(* Logix 5000 project; controller cal1632 1756-L62 rev 16.20; software revision 16.05; part 32 of 61 *)
(* tags used below, declared in another part *)
   FAULT : BOOL;
   HMI : BOOL;
   p01_recipe_active : recipe;
   p01r09 : routine;
   p01r09_pb_global_reset : BOOL;
   p01r13_line_running : BOOL;
   p02_dint_from_hmi : hmi_dint;
   p20_di_acc_empty : BOOL;
   p20_do_close_nip : BOOL;
   p20_do_engage_lfr_clutch : BOOL;
   p21_di_close_exit_clamp : BOOL;
   p21_di_close_inlet_clamp : BOOL;
   p21_di_open_splice_platen : BOOL;
   p21_di_platen_not_closed : BOOL;
   p21_di_splice_2_hand_close : BOOL;
   p21_dint_to_hmi : DINT[16];
   p21_do_close_exit_clamp_sv : BOOL;
   p21_do_close_inlet_clamp_sv : BOOL;
   p21_do_close_platen_sv : BOOL;
   p21r07 : routine;
   p21r07_timer_fault : TIMER[4];
   p21r07_timer_warning : TIMER[4];
   p21r08 : routine;
   p21r08_timer_fault : TIMER[4];
   p21r08_timer_warning : TIMER[4];
   p21r09 : routine;
   p21r09_timer_fault : TIMER[4];
   p21r09_timer_warning : TIMER[4];
   p21r10 : routine;
   p21r10_permissive_run : BOOL;
   p21r10_remaining_cure_time : DINT;
   p21r10_remaining_cure_time_sec : REAL;
   p21r10_splice_press_1 : SYS_ENC;
   p21r10_state : DINT;
   p21r10_status : DINT;
   p21r10_timer_exit_open_delay : TIMER;
   p21r10_timer_fault : TIMER[4];
   p21r10_timer_inlet_open_delay : TIMER;
   p21r10_timer_platen_open_delay : TIMER;
   p21r10_timer_press_cure : TIMER;
   p21r10_timer_warning : TIMER[4];
   p21r16 : routine;
(* P21_Splice_Press, continued *)

ROUTINE R07_Alarms   (* ladder *)
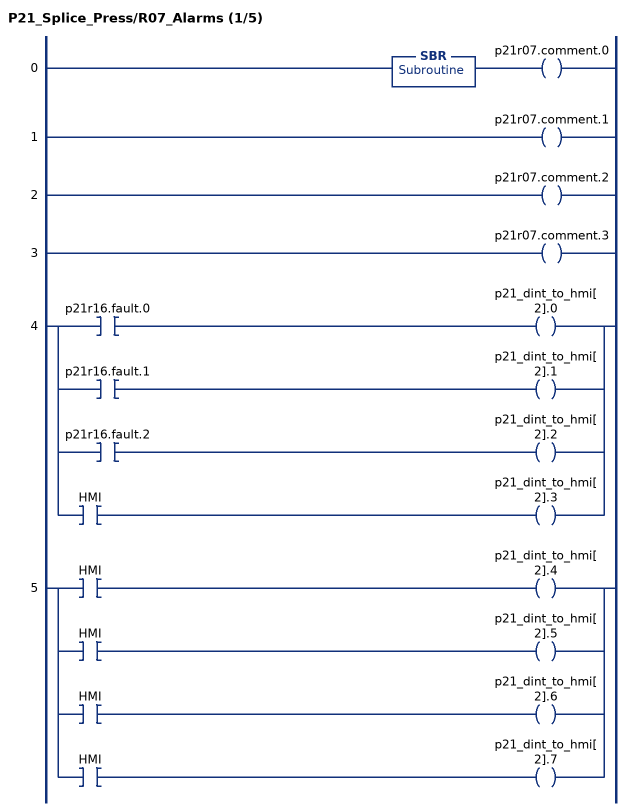
   0: SBR()OTE(p21r07.comment.0);
   1: OTE(p21r07.comment.1);
   2: OTE(p21r07.comment.2);
   3: OTE(p21r07.comment.3);
   4: [XIC(p21r16.fault.0) OTE(p21_dint_to_hmi[2].0) ,XIC(p21r16.fault.1) OTE(p21_dint_to_hmi[2].1) ,XIC(p21r16.fault.2) OTE(p21_dint_to_hmi[2].2) ,XIC(HMI) OTE(p21_dint_to_hmi[2].3) ];
   5: [XIC(HMI) OTE(p21_dint_to_hmi[2].4) ,XIC(HMI) OTE(p21_dint_to_hmi[2].5) ,XIC(HMI) OTE(p21_dint_to_hmi[2].6) ,XIC(HMI) OTE(p21_dint_to_hmi[2].7) ];
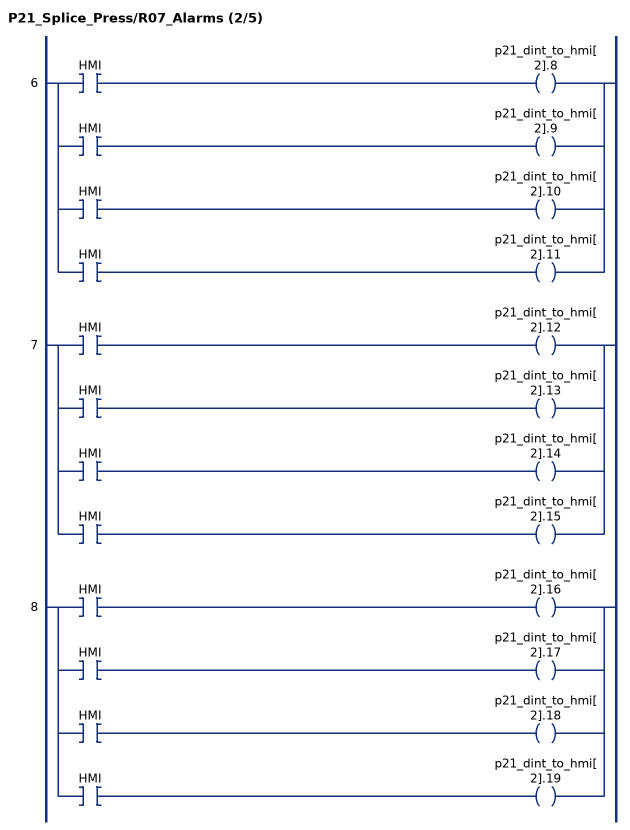
   6: [XIC(HMI) OTE(p21_dint_to_hmi[2].8) ,XIC(HMI) OTE(p21_dint_to_hmi[2].9) ,XIC(HMI) OTE(p21_dint_to_hmi[2].10) ,XIC(HMI) OTE(p21_dint_to_hmi[2].11) ];
   7: [XIC(HMI) OTE(p21_dint_to_hmi[2].12) ,XIC(HMI) OTE(p21_dint_to_hmi[2].13) ,XIC(HMI) OTE(p21_dint_to_hmi[2].14) ,XIC(HMI) OTE(p21_dint_to_hmi[2].15) ];
   8: [XIC(HMI) OTE(p21_dint_to_hmi[2].16) ,XIC(HMI) OTE(p21_dint_to_hmi[2].17) ,XIC(HMI) OTE(p21_dint_to_hmi[2].18) ,XIC(HMI) OTE(p21_dint_to_hmi[2].19) ];
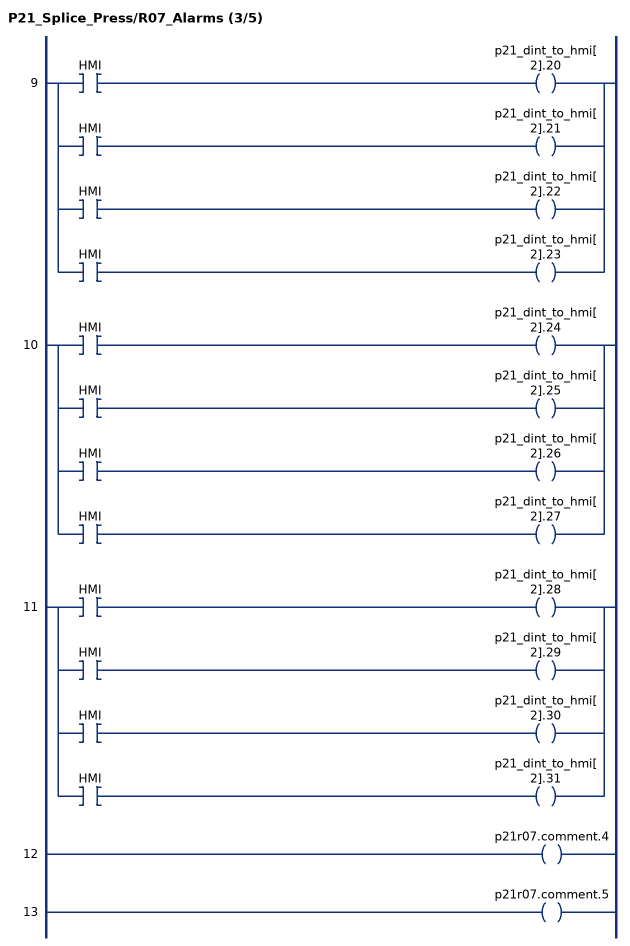
   9: [XIC(HMI) OTE(p21_dint_to_hmi[2].20) ,XIC(HMI) OTE(p21_dint_to_hmi[2].21) ,XIC(HMI) OTE(p21_dint_to_hmi[2].22) ,XIC(HMI) OTE(p21_dint_to_hmi[2].23) ];
   10: [XIC(HMI) OTE(p21_dint_to_hmi[2].24) ,XIC(HMI) OTE(p21_dint_to_hmi[2].25) ,XIC(HMI) OTE(p21_dint_to_hmi[2].26) ,XIC(HMI) OTE(p21_dint_to_hmi[2].27) ];
   11: [XIC(HMI) OTE(p21_dint_to_hmi[2].28) ,XIC(HMI) OTE(p21_dint_to_hmi[2].29) ,XIC(HMI) OTE(p21_dint_to_hmi[2].30) ,XIC(HMI) OTE(p21_dint_to_hmi[2].31) ];
   12: OTE(p21r07.comment.4);
   13: OTE(p21r07.comment.5);
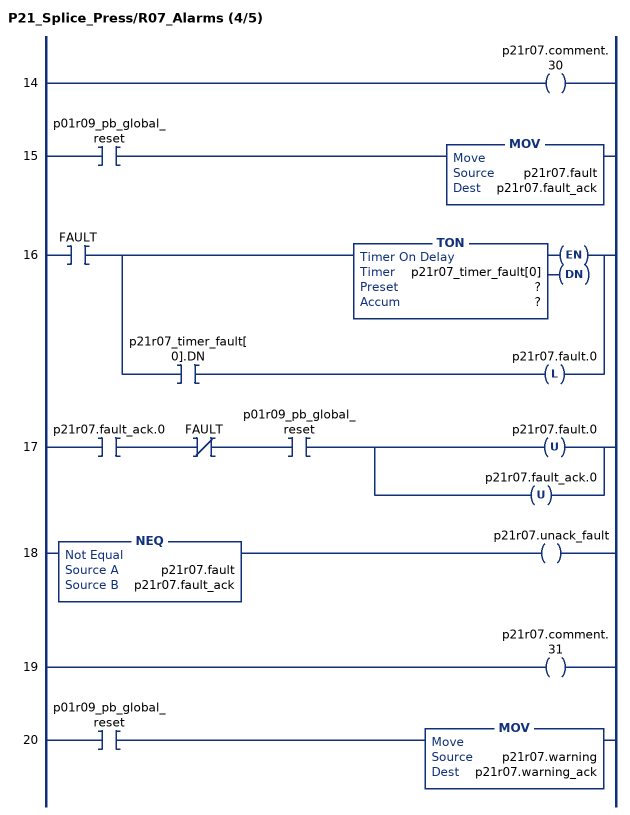
   14: OTE(p21r07.comment.30);
   15: XIC(p01r09_pb_global_reset)MOV(p21r07.fault,p21r07.fault_ack);
   16: XIC(FAULT)[TON(p21r07_timer_fault[0],?,?) ,XIC(p21r07_timer_fault[0].DN) OTL(p21r07.fault.0) ];
   17: XIC(p21r07.fault_ack.0)XIO(FAULT)XIC(p01r09_pb_global_reset)[OTU(p21r07.fault.0) ,OTU(p21r07.fault_ack.0) ];
   18: NEQ(p21r07.fault,p21r07.fault_ack)OTE(p21r07.unack_fault);
   19: OTE(p21r07.comment.31);
   20: XIC(p01r09_pb_global_reset)MOV(p21r07.warning,p21r07.warning_ack);
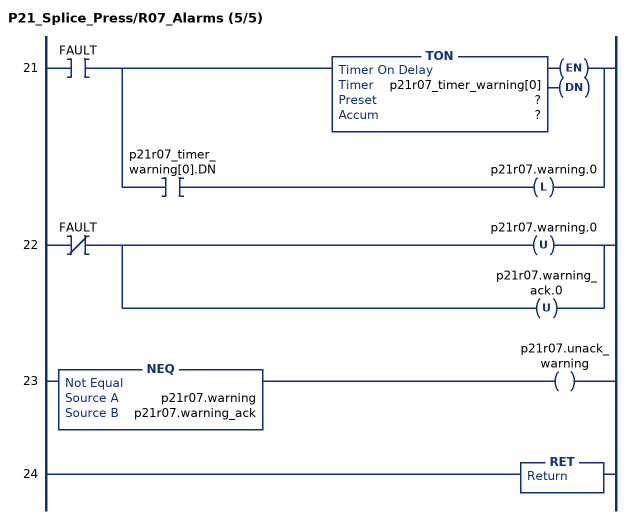
   21: XIC(FAULT)[TON(p21r07_timer_warning[0],?,?) ,XIC(p21r07_timer_warning[0].DN) OTL(p21r07.warning.0) ];
   22: XIO(FAULT)[OTU(p21r07.warning.0) ,OTU(p21r07.warning_ack.0) ];
   23: NEQ(p21r07.warning,p21r07.warning_ack)OTE(p21r07.unack_warning);
   24: RET();
END_ROUTINE

ROUTINE R08_Warnings   (* ladder *)
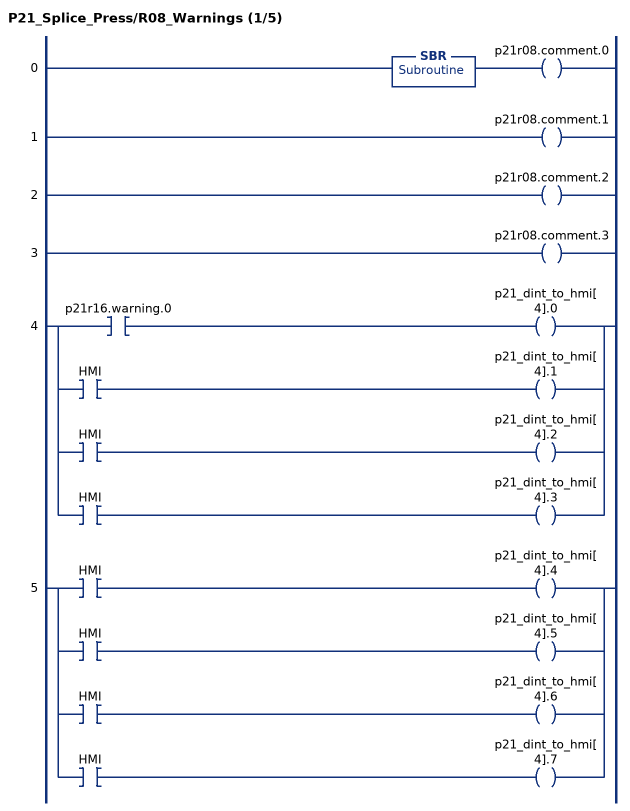
   0: SBR()OTE(p21r08.comment.0);
   1: OTE(p21r08.comment.1);
   2: OTE(p21r08.comment.2);
   3: OTE(p21r08.comment.3);
   4: [XIC(p21r16.warning.0) OTE(p21_dint_to_hmi[4].0) ,XIC(HMI) OTE(p21_dint_to_hmi[4].1) ,XIC(HMI) OTE(p21_dint_to_hmi[4].2) ,XIC(HMI) OTE(p21_dint_to_hmi[4].3) ];
   5: [XIC(HMI) OTE(p21_dint_to_hmi[4].4) ,XIC(HMI) OTE(p21_dint_to_hmi[4].5) ,XIC(HMI) OTE(p21_dint_to_hmi[4].6) ,XIC(HMI) OTE(p21_dint_to_hmi[4].7) ];
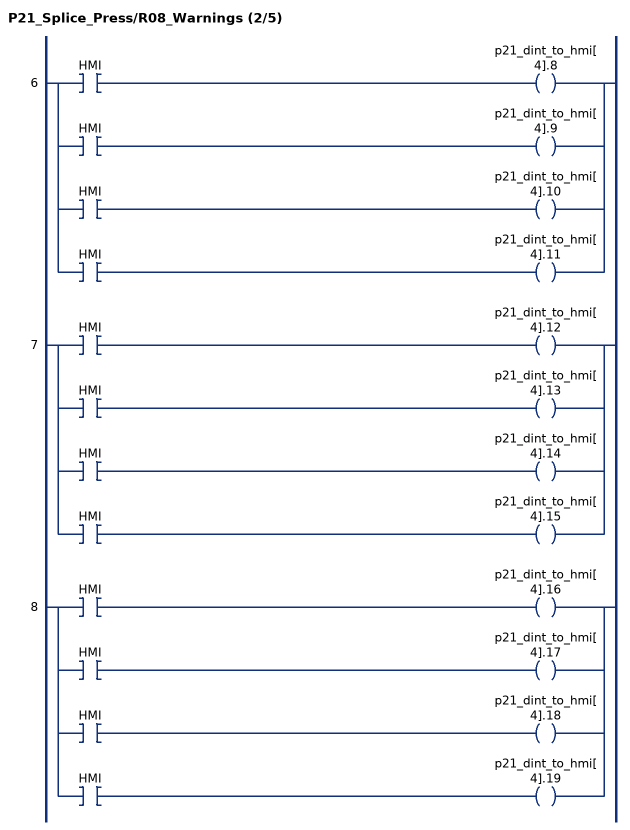
   6: [XIC(HMI) OTE(p21_dint_to_hmi[4].8) ,XIC(HMI) OTE(p21_dint_to_hmi[4].9) ,XIC(HMI) OTE(p21_dint_to_hmi[4].10) ,XIC(HMI) OTE(p21_dint_to_hmi[4].11) ];
   7: [XIC(HMI) OTE(p21_dint_to_hmi[4].12) ,XIC(HMI) OTE(p21_dint_to_hmi[4].13) ,XIC(HMI) OTE(p21_dint_to_hmi[4].14) ,XIC(HMI) OTE(p21_dint_to_hmi[4].15) ];
   8: [XIC(HMI) OTE(p21_dint_to_hmi[4].16) ,XIC(HMI) OTE(p21_dint_to_hmi[4].17) ,XIC(HMI) OTE(p21_dint_to_hmi[4].18) ,XIC(HMI) OTE(p21_dint_to_hmi[4].19) ];
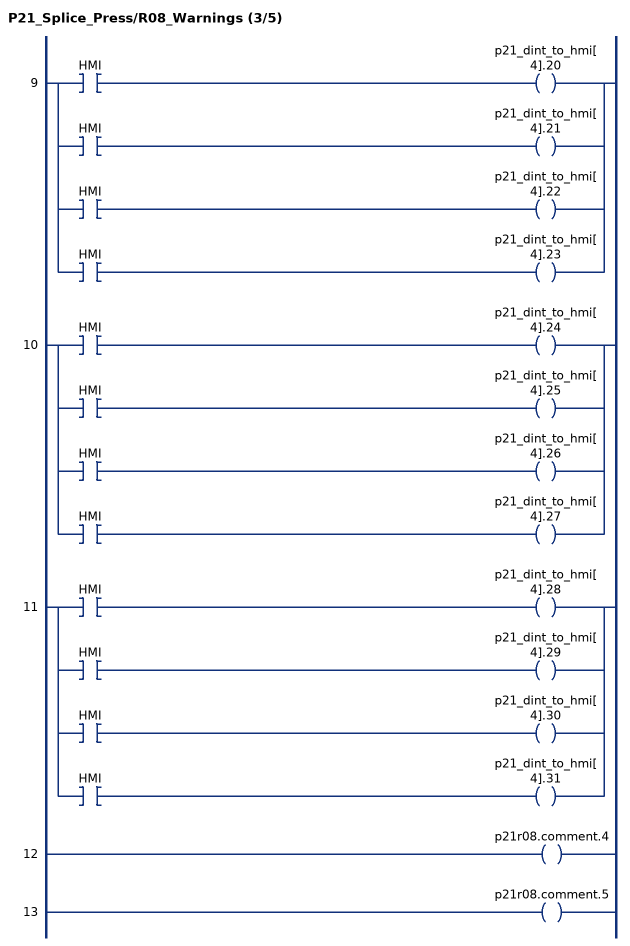
   9: [XIC(HMI) OTE(p21_dint_to_hmi[4].20) ,XIC(HMI) OTE(p21_dint_to_hmi[4].21) ,XIC(HMI) OTE(p21_dint_to_hmi[4].22) ,XIC(HMI) OTE(p21_dint_to_hmi[4].23) ];
   10: [XIC(HMI) OTE(p21_dint_to_hmi[4].24) ,XIC(HMI) OTE(p21_dint_to_hmi[4].25) ,XIC(HMI) OTE(p21_dint_to_hmi[4].26) ,XIC(HMI) OTE(p21_dint_to_hmi[4].27) ];
   11: [XIC(HMI) OTE(p21_dint_to_hmi[4].28) ,XIC(HMI) OTE(p21_dint_to_hmi[4].29) ,XIC(HMI) OTE(p21_dint_to_hmi[4].30) ,XIC(HMI) OTE(p21_dint_to_hmi[4].31) ];
   12: OTE(p21r08.comment.4);
   13: OTE(p21r08.comment.5);
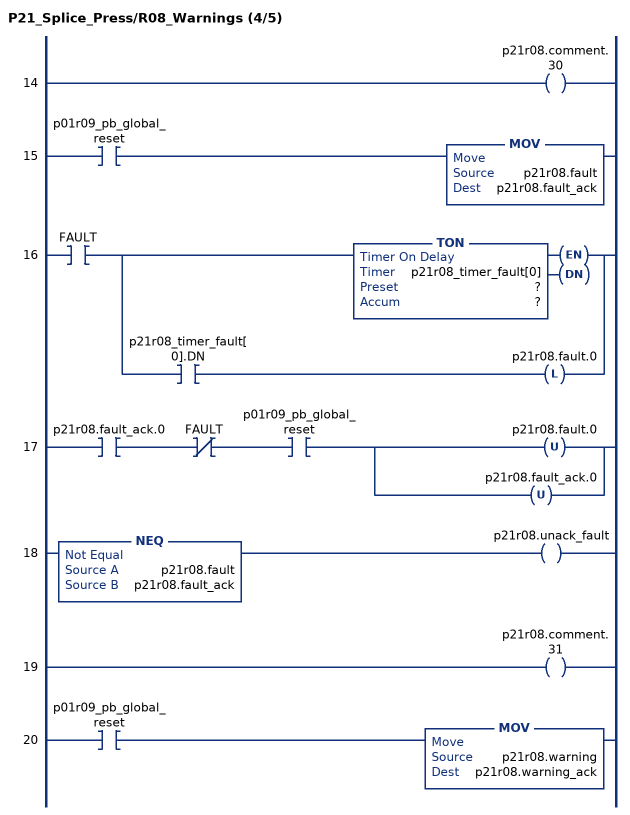
   14: OTE(p21r08.comment.30);
   15: XIC(p01r09_pb_global_reset)MOV(p21r08.fault,p21r08.fault_ack);
   16: XIC(FAULT)[TON(p21r08_timer_fault[0],?,?) ,XIC(p21r08_timer_fault[0].DN) OTL(p21r08.fault.0) ];
   17: XIC(p21r08.fault_ack.0)XIO(FAULT)XIC(p01r09_pb_global_reset)[OTU(p21r08.fault.0) ,OTU(p21r08.fault_ack.0) ];
   18: NEQ(p21r08.fault,p21r08.fault_ack)OTE(p21r08.unack_fault);
   19: OTE(p21r08.comment.31);
   20: XIC(p01r09_pb_global_reset)MOV(p21r08.warning,p21r08.warning_ack);
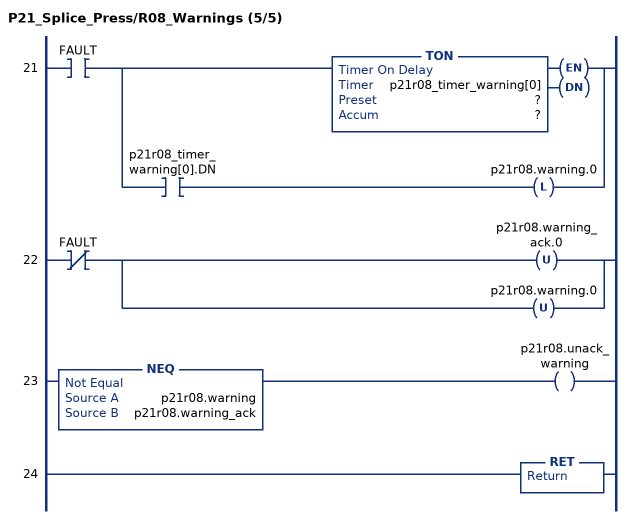
   21: XIC(FAULT)[TON(p21r08_timer_warning[0],?,?) ,XIC(p21r08_timer_warning[0].DN) OTL(p21r08.warning.0) ];
   22: XIO(FAULT)[OTU(p21r08.warning_ack.0) ,OTU(p21r08.warning.0) ];
   23: NEQ(p21r08.warning,p21r08.warning_ack)OTE(p21r08.unack_warning);
   24: RET();
END_ROUTINE

ROUTINE R09_Modes   (* ladder *)
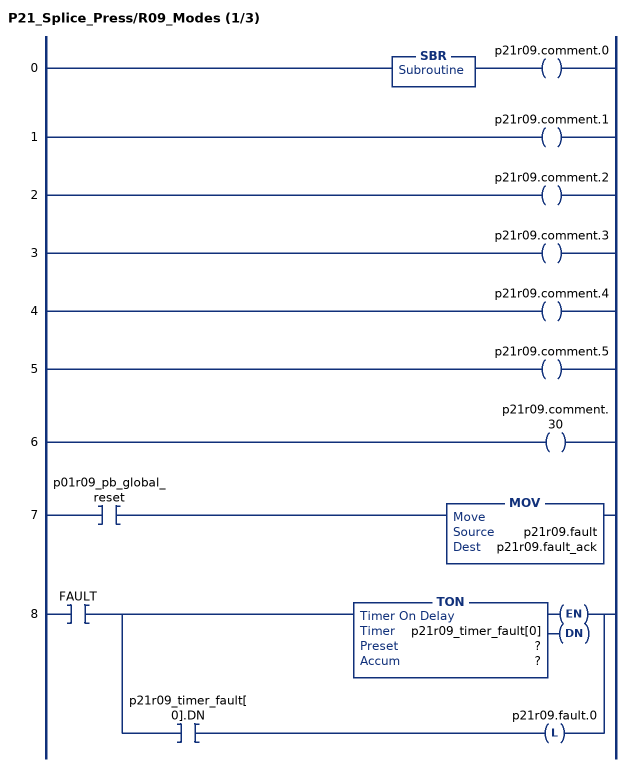
   0: SBR()OTE(p21r09.comment.0);
   1: OTE(p21r09.comment.1);
   2: OTE(p21r09.comment.2);
   3: OTE(p21r09.comment.3);
   4: OTE(p21r09.comment.4);
   5: OTE(p21r09.comment.5);
   6: OTE(p21r09.comment.30);
   7: XIC(p01r09_pb_global_reset)MOV(p21r09.fault,p21r09.fault_ack);
   8: XIC(FAULT)[TON(p21r09_timer_fault[0],?,?) ,XIC(p21r09_timer_fault[0].DN) OTL(p21r09.fault.0) ];
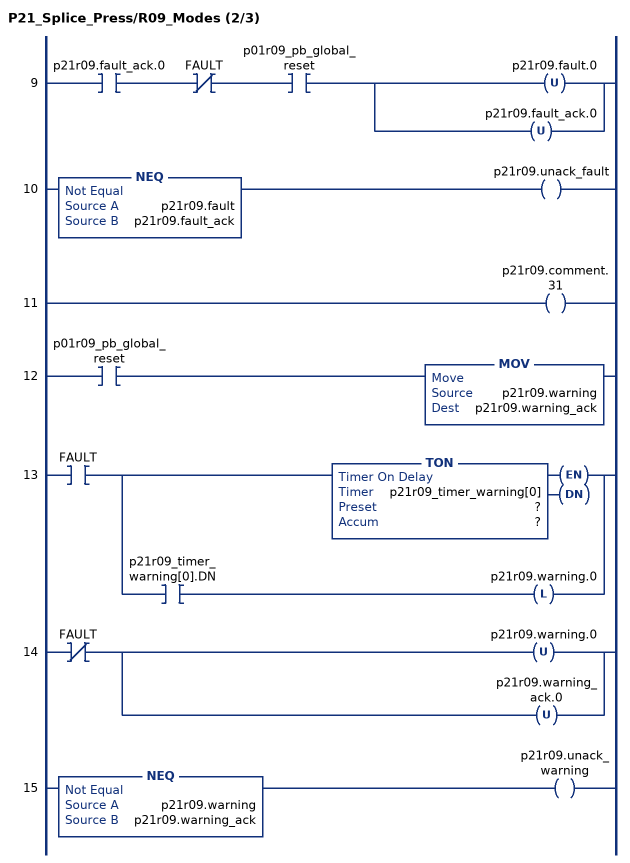
   9: XIC(p21r09.fault_ack.0)XIO(FAULT)XIC(p01r09_pb_global_reset)[OTU(p21r09.fault.0) ,OTU(p21r09.fault_ack.0) ];
   10: NEQ(p21r09.fault,p21r09.fault_ack)OTE(p21r09.unack_fault);
   11: OTE(p21r09.comment.31);
   12: XIC(p01r09_pb_global_reset)MOV(p21r09.warning,p21r09.warning_ack);
   13: XIC(FAULT)[TON(p21r09_timer_warning[0],?,?) ,XIC(p21r09_timer_warning[0].DN) OTL(p21r09.warning.0) ];
   14: XIO(FAULT)[OTU(p21r09.warning.0) ,OTU(p21r09.warning_ack.0) ];
   15: NEQ(p21r09.warning,p21r09.warning_ack)OTE(p21r09.unack_warning);
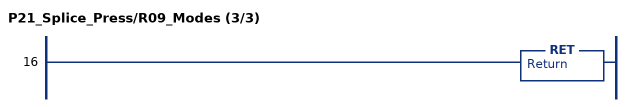
   16: RET();
END_ROUTINE

ROUTINE R10_Sequence   (* ladder *)
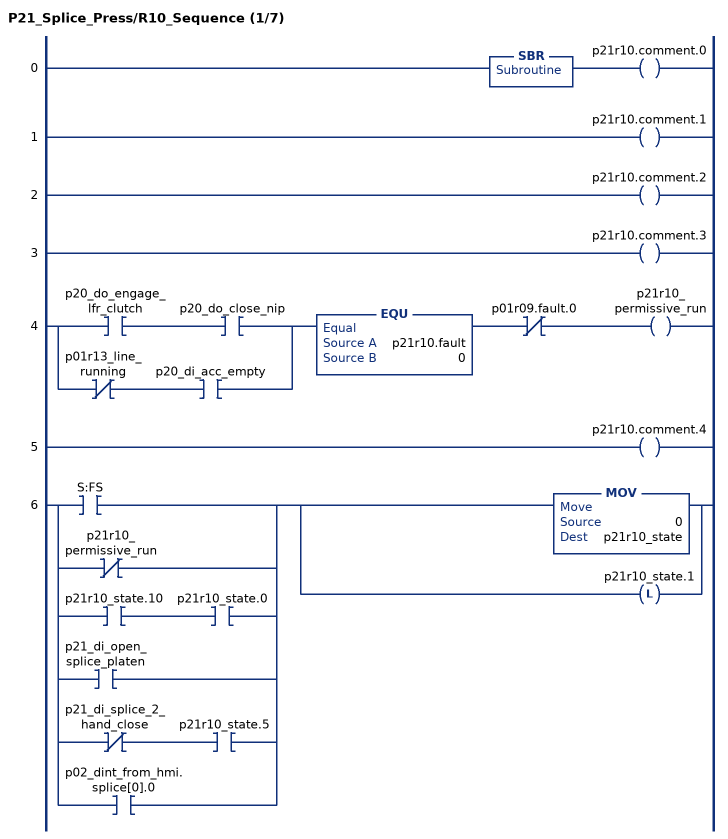
   0: SBR()OTE(p21r10.comment.0);
   1: OTE(p21r10.comment.1);
   2: OTE(p21r10.comment.2);
   3: OTE(p21r10.comment.3);
   4: [XIC(p20_do_engage_lfr_clutch) XIC(p20_do_close_nip) ,XIO(p01r13_line_running) XIC(p20_di_acc_empty) ]EQU(p21r10.fault,0)XIO(p01r09.fault.0)OTE(p21r10_permissive_run);
   5: OTE(p21r10.comment.4);
   6: [XIC(S:FS) ,XIO(p21r10_permissive_run) ,XIC(p21r10_state.10) XIC(p21r10_state.0) ,XIC(p21_di_open_splice_platen) ,XIO(p21_di_splice_2_hand_close) XIC(p21r10_state.5) ,XIC(p02_dint_from_hmi.splice[0].0) ][MOV(0,p21r10_state) ,OTL(p21r10_state.1) ];
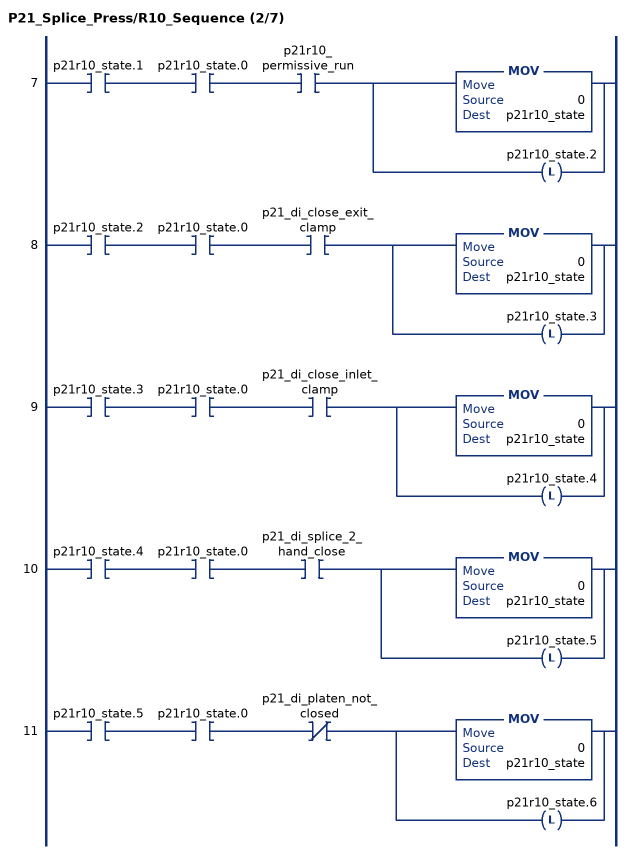
   7: XIC(p21r10_state.1)XIC(p21r10_state.0)XIC(p21r10_permissive_run)[MOV(0,p21r10_state) ,OTL(p21r10_state.2) ];
   8: XIC(p21r10_state.2)XIC(p21r10_state.0)XIC(p21_di_close_exit_clamp)[MOV(0,p21r10_state) ,OTL(p21r10_state.3) ];
   9: XIC(p21r10_state.3)XIC(p21r10_state.0)XIC(p21_di_close_inlet_clamp)[MOV(0,p21r10_state) ,OTL(p21r10_state.4) ];
   10: XIC(p21r10_state.4)XIC(p21r10_state.0)XIC(p21_di_splice_2_hand_close)[MOV(0,p21r10_state) ,OTL(p21r10_state.5) ];
   11: XIC(p21r10_state.5)XIC(p21r10_state.0)XIO(p21_di_platen_not_closed)[MOV(0,p21r10_state) ,OTL(p21r10_state.6) ];
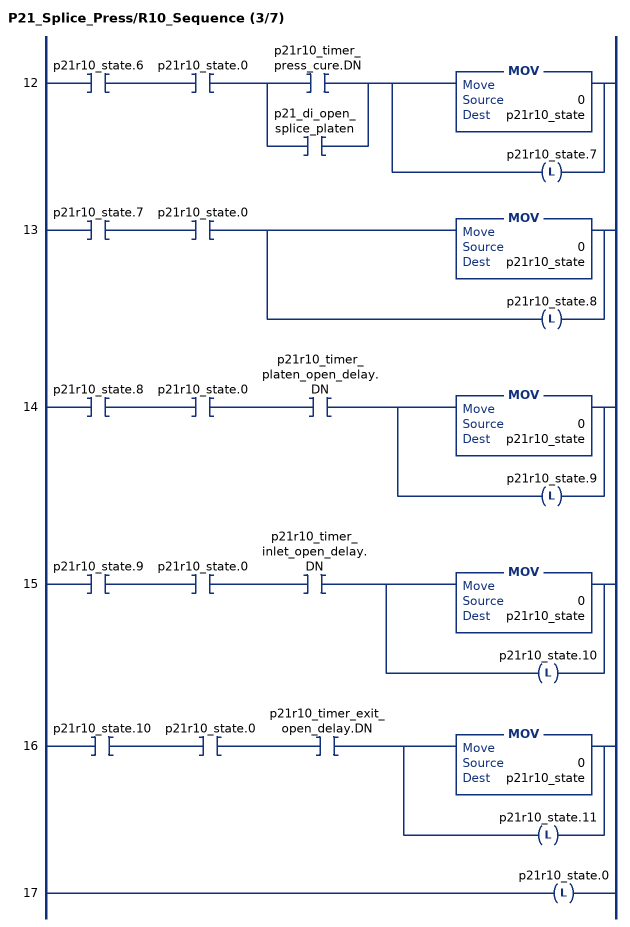
   12: XIC(p21r10_state.6)XIC(p21r10_state.0)[XIC(p21r10_timer_press_cure.DN) ,XIC(p21_di_open_splice_platen) ][MOV(0,p21r10_state) ,OTL(p21r10_state.7) ];
   13: XIC(p21r10_state.7)XIC(p21r10_state.0)[MOV(0,p21r10_state) ,OTL(p21r10_state.8) ];
   14: XIC(p21r10_state.8)XIC(p21r10_state.0)XIC(p21r10_timer_platen_open_delay.DN)[MOV(0,p21r10_state) ,OTL(p21r10_state.9) ];
   15: XIC(p21r10_state.9)XIC(p21r10_state.0)XIC(p21r10_timer_inlet_open_delay.DN)[MOV(0,p21r10_state) ,OTL(p21r10_state.10) ];
   16: XIC(p21r10_state.10)XIC(p21r10_state.0)XIC(p21r10_timer_exit_open_delay.DN)[MOV(0,p21r10_state) ,OTL(p21r10_state.11) ];
   17: OTL(p21r10_state.0);
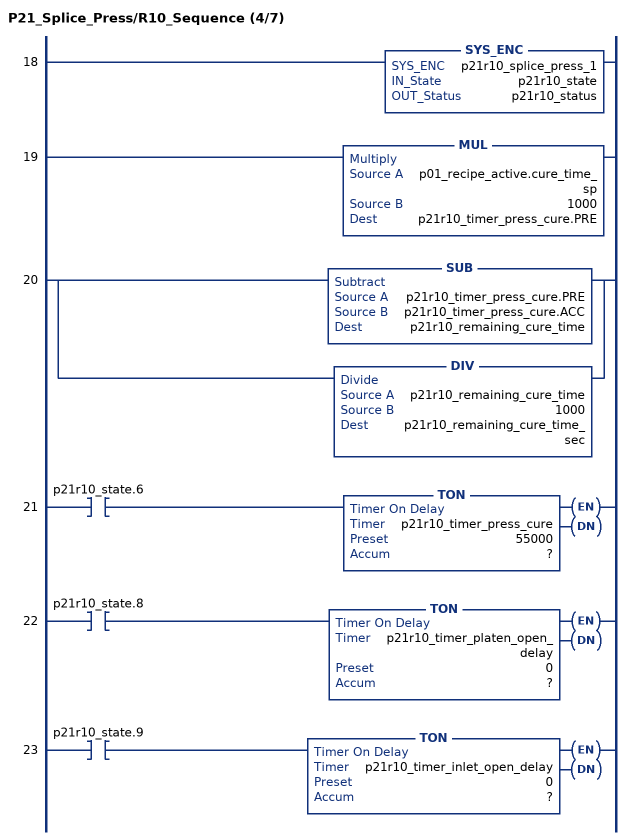
   18: SYS_ENC(p21r10_splice_press_1,p21r10_state,p21r10_status);
   19: MUL(p01_recipe_active.cure_time_sp,1000,p21r10_timer_press_cure.PRE);
   20: [SUB(p21r10_timer_press_cure.PRE,p21r10_timer_press_cure.ACC,p21r10_remaining_cure_time) ,DIV(p21r10_remaining_cure_time,1000,p21r10_remaining_cure_time_sec) ];
   21: XIC(p21r10_state.6)TON(p21r10_timer_press_cure,?,?);
   22: XIC(p21r10_state.8)TON(p21r10_timer_platen_open_delay,?,?);
   23: XIC(p21r10_state.9)TON(p21r10_timer_inlet_open_delay,?,?);
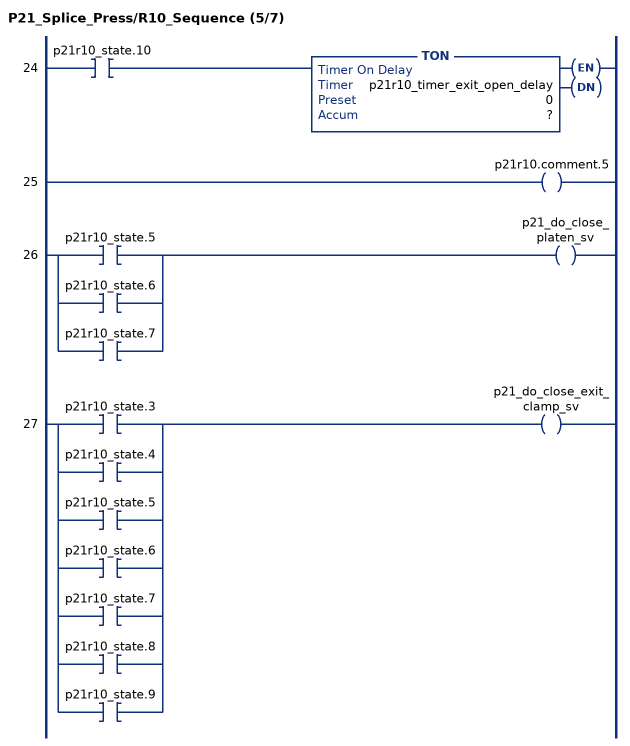
   24: XIC(p21r10_state.10)TON(p21r10_timer_exit_open_delay,?,?);
   25: OTE(p21r10.comment.5);
   26: [XIC(p21r10_state.5) ,XIC(p21r10_state.6) ,XIC(p21r10_state.7) ]OTE(p21_do_close_platen_sv);
   27: [XIC(p21r10_state.3) ,XIC(p21r10_state.4) ,XIC(p21r10_state.5) ,XIC(p21r10_state.6) ,XIC(p21r10_state.7) ,XIC(p21r10_state.8) ,XIC(p21r10_state.9) ]OTE(p21_do_close_exit_clamp_sv);
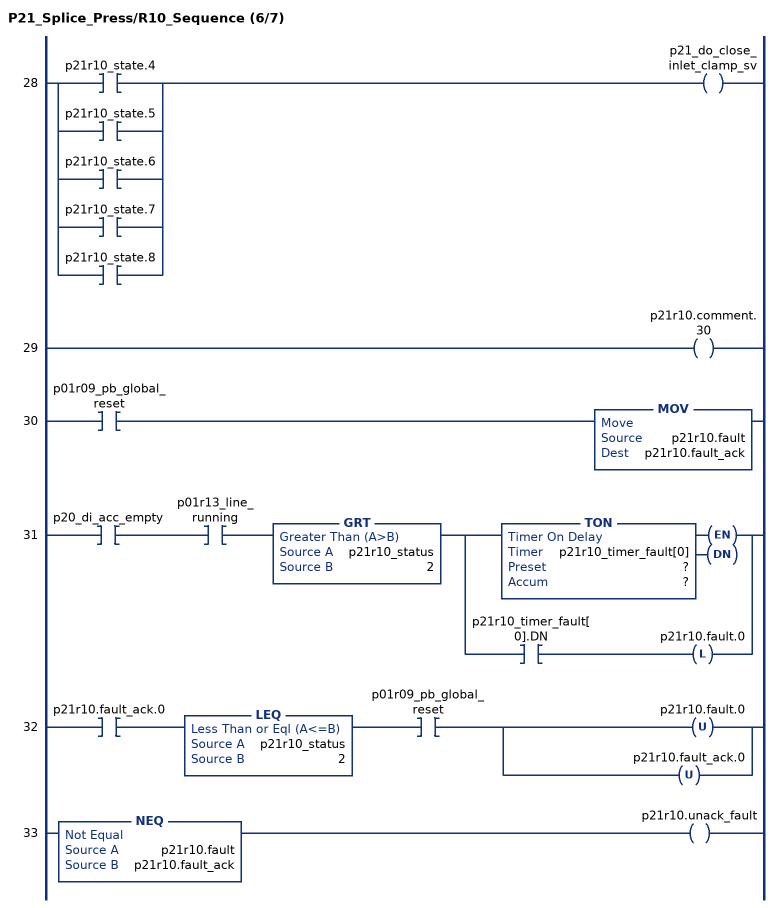
   28: [XIC(p21r10_state.4) ,XIC(p21r10_state.5) ,XIC(p21r10_state.6) ,XIC(p21r10_state.7) ,XIC(p21r10_state.8) ]OTE(p21_do_close_inlet_clamp_sv);
   29: OTE(p21r10.comment.30);
   30: XIC(p01r09_pb_global_reset)MOV(p21r10.fault,p21r10.fault_ack);
   31: XIC(p20_di_acc_empty)XIC(p01r13_line_running)GRT(p21r10_status,2)[TON(p21r10_timer_fault[0],?,?) ,XIC(p21r10_timer_fault[0].DN) OTL(p21r10.fault.0) ];
   32: XIC(p21r10.fault_ack.0)LEQ(p21r10_status,2)XIC(p01r09_pb_global_reset)[OTU(p21r10.fault.0) ,OTU(p21r10.fault_ack.0) ];
   33: NEQ(p21r10.fault,p21r10.fault_ack)OTE(p21r10.unack_fault);
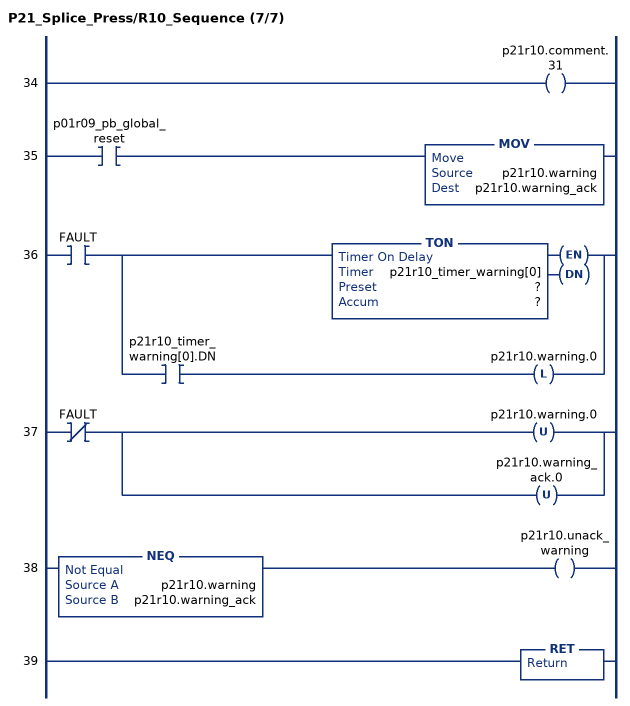
   34: OTE(p21r10.comment.31);
   35: XIC(p01r09_pb_global_reset)MOV(p21r10.warning,p21r10.warning_ack);
   36: XIC(FAULT)[TON(p21r10_timer_warning[0],?,?) ,XIC(p21r10_timer_warning[0].DN) OTL(p21r10.warning.0) ];
   37: XIO(FAULT)[OTU(p21r10.warning.0) ,OTU(p21r10.warning_ack.0) ];
   38: NEQ(p21r10.warning,p21r10.warning_ack)OTE(p21r10.unack_warning);
   39: RET();
END_ROUTINE
